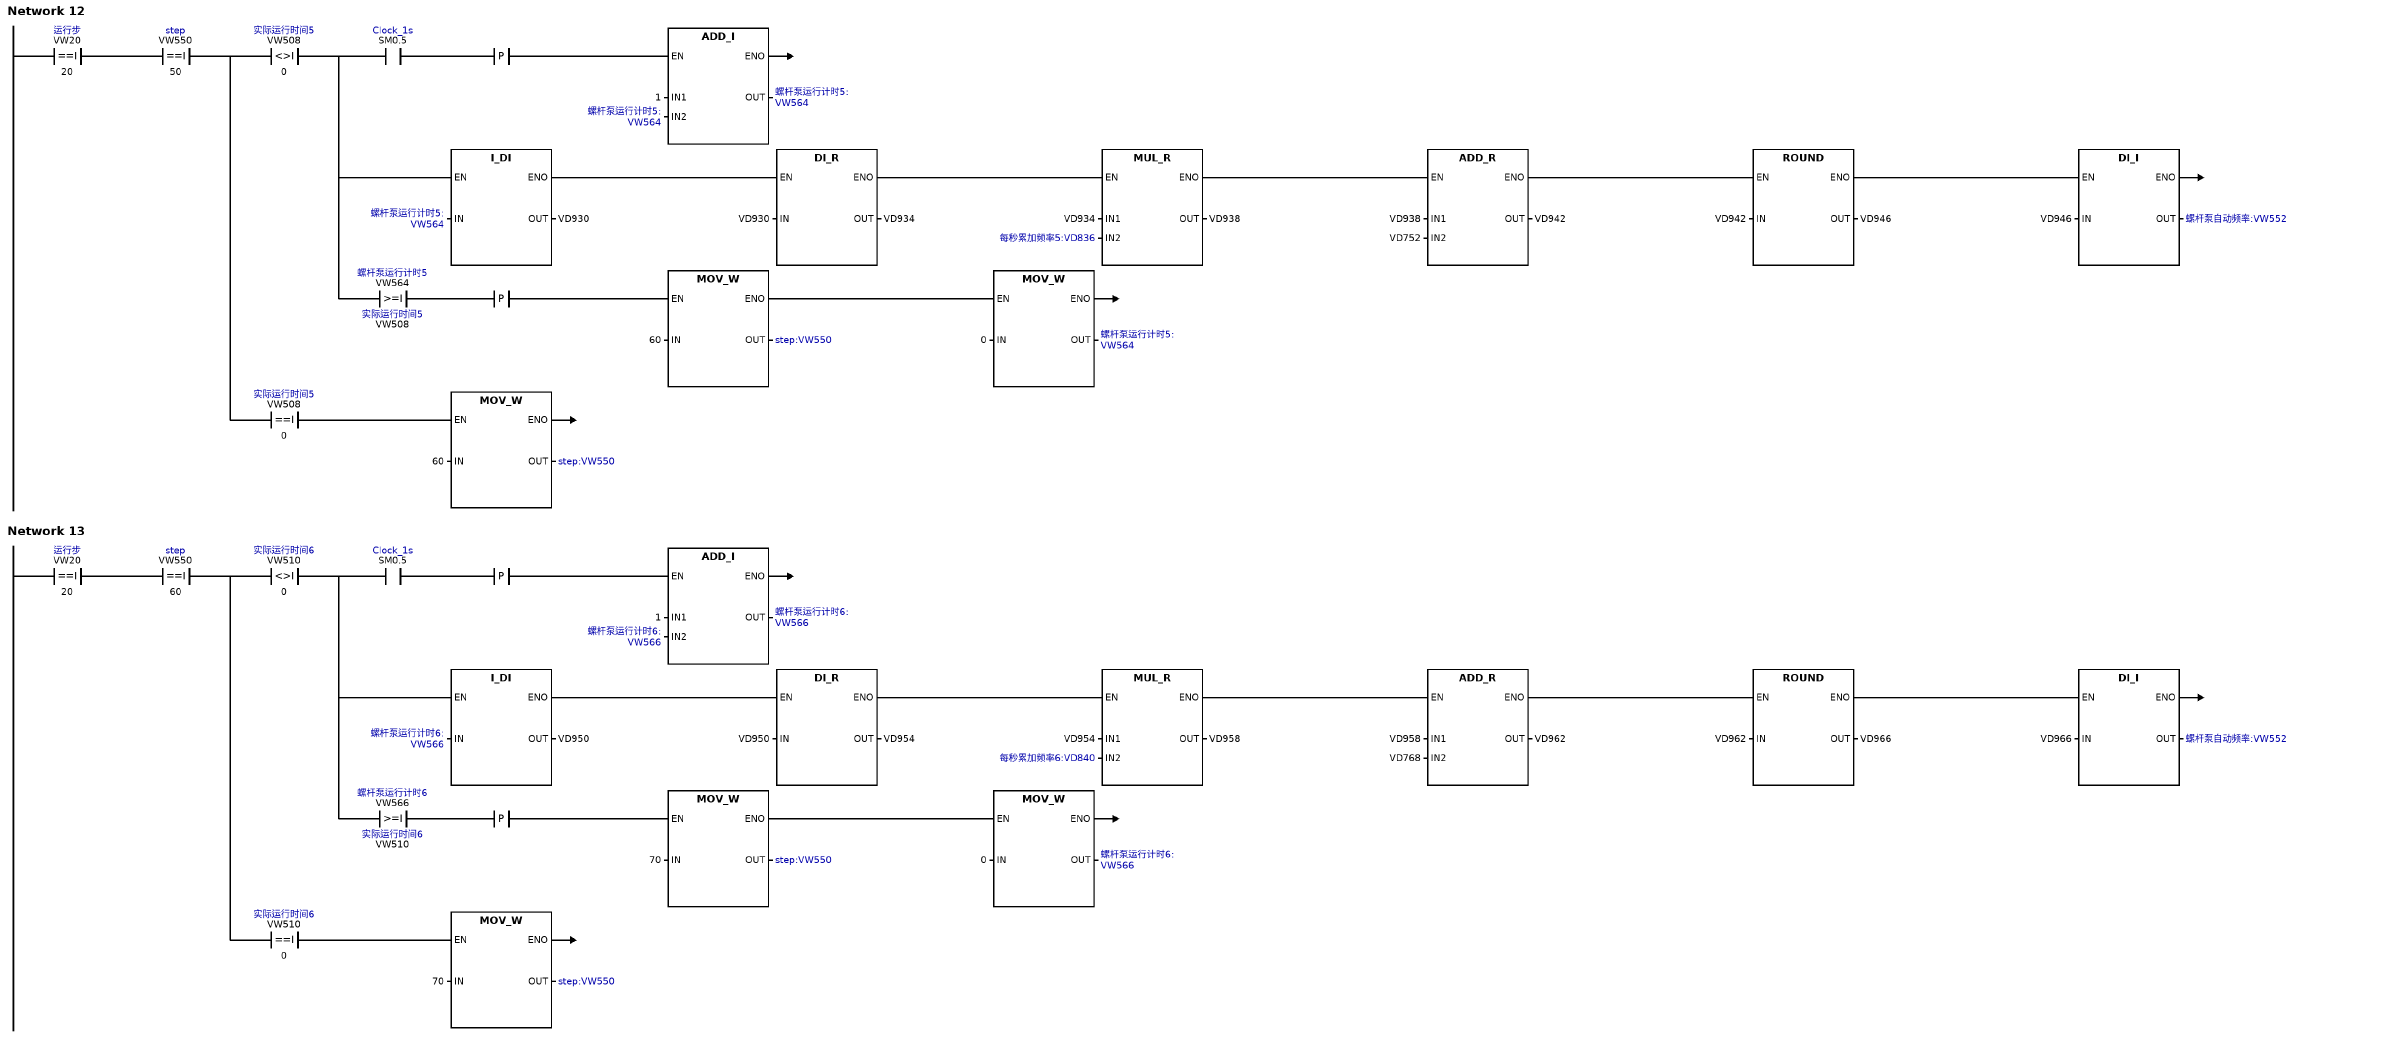
[picture p24: SBR4 networks 12-13]
Network 12
LDW=   运行步:VW20, 20
AW=    step:VW550, 50
LPS
AW<>   实际运行时间5:VW508, 0
LPS
A      Clock_1s:SM0.5
EU
+I     1, 螺杆泵运行计时5:VW564
LRD
ITD    螺杆泵运行计时5:VW564, VD930
AENO
DTR    VD930, VD934
AENO
MOVR   VD934, VD938
AENO
*R     每秒累加频率5:VD836, VD938
AENO
MOVR   VD938, VD942
AENO
+R     VD752, VD942
AENO
ROUND  VD942, VD946
AENO
DTI    VD946, 螺杆泵自动频率:VW552
LPP
AW>=   螺杆泵运行计时5:VW564, 实际运行时间5:VW508
EU
MOVW   60, step:VW550
AENO
MOVW   0, 螺杆泵运行计时5:VW564
LPP
AW=    实际运行时间5:VW508, 0
MOVW   60, step:VW550
Network 13
LDW=   运行步:VW20, 20
AW=    step:VW550, 60
LPS
AW<>   实际运行时间6:VW510, 0
LPS
A      Clock_1s:SM0.5
EU
+I     1, 螺杆泵运行计时6:VW566
LRD
ITD    螺杆泵运行计时6:VW566, VD950
AENO
DTR    VD950, VD954
AENO
MOVR   VD954, VD958
AENO
*R     每秒累加频率6:VD840, VD958
AENO
MOVR   VD958, VD962
AENO
+R     VD768, VD962
AENO
ROUND  VD962, VD966
AENO
DTI    VD966, 螺杆泵自动频率:VW552
LPP
AW>=   螺杆泵运行计时6:VW566, 实际运行时间6:VW510
EU
MOVW   70, step:VW550
AENO
MOVW   0, 螺杆泵运行计时6:VW566
LPP
AW=    实际运行时间6:VW510, 0
MOVW   70, step:VW550
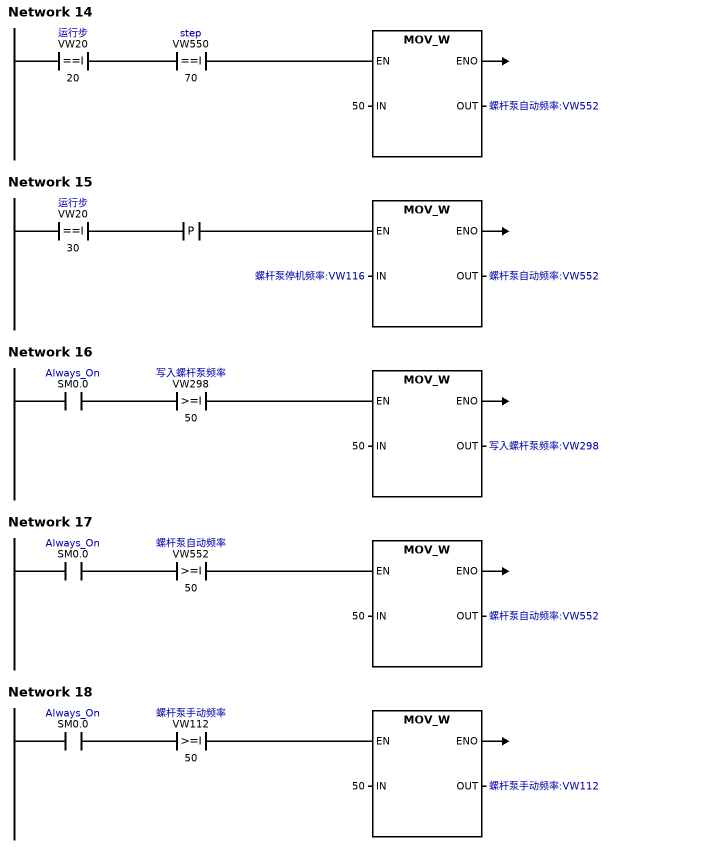
Network 14
LDW=   运行步:VW20, 20
AW=    step:VW550, 70
MOVW   50, 螺杆泵自动频率:VW552
Network 15
LDW=   运行步:VW20, 30
EU
MOVW   螺杆泵停机频率:VW116, 螺杆泵自动频率:VW552
Network 16
LD     Always_On:SM0.0
AW>=   写入螺杆泵频率:VW298, 50
MOVW   50, 写入螺杆泵频率:VW298
Network 17
LD     Always_On:SM0.0
AW>=   螺杆泵自动频率:VW552, 50
MOVW   50, 螺杆泵自动频率:VW552
Network 18
LD     Always_On:SM0.0
AW>=   螺杆泵手动频率:VW112, 50
MOVW   50, 螺杆泵手动频率:VW112
Network 19
// ‘////////////////////////////
END_SUBROUTINE_BLOCK

SUBROUTINE_BLOCK 罗茨泵PID:SBR5
TITLE=子程序注释
BEGIN
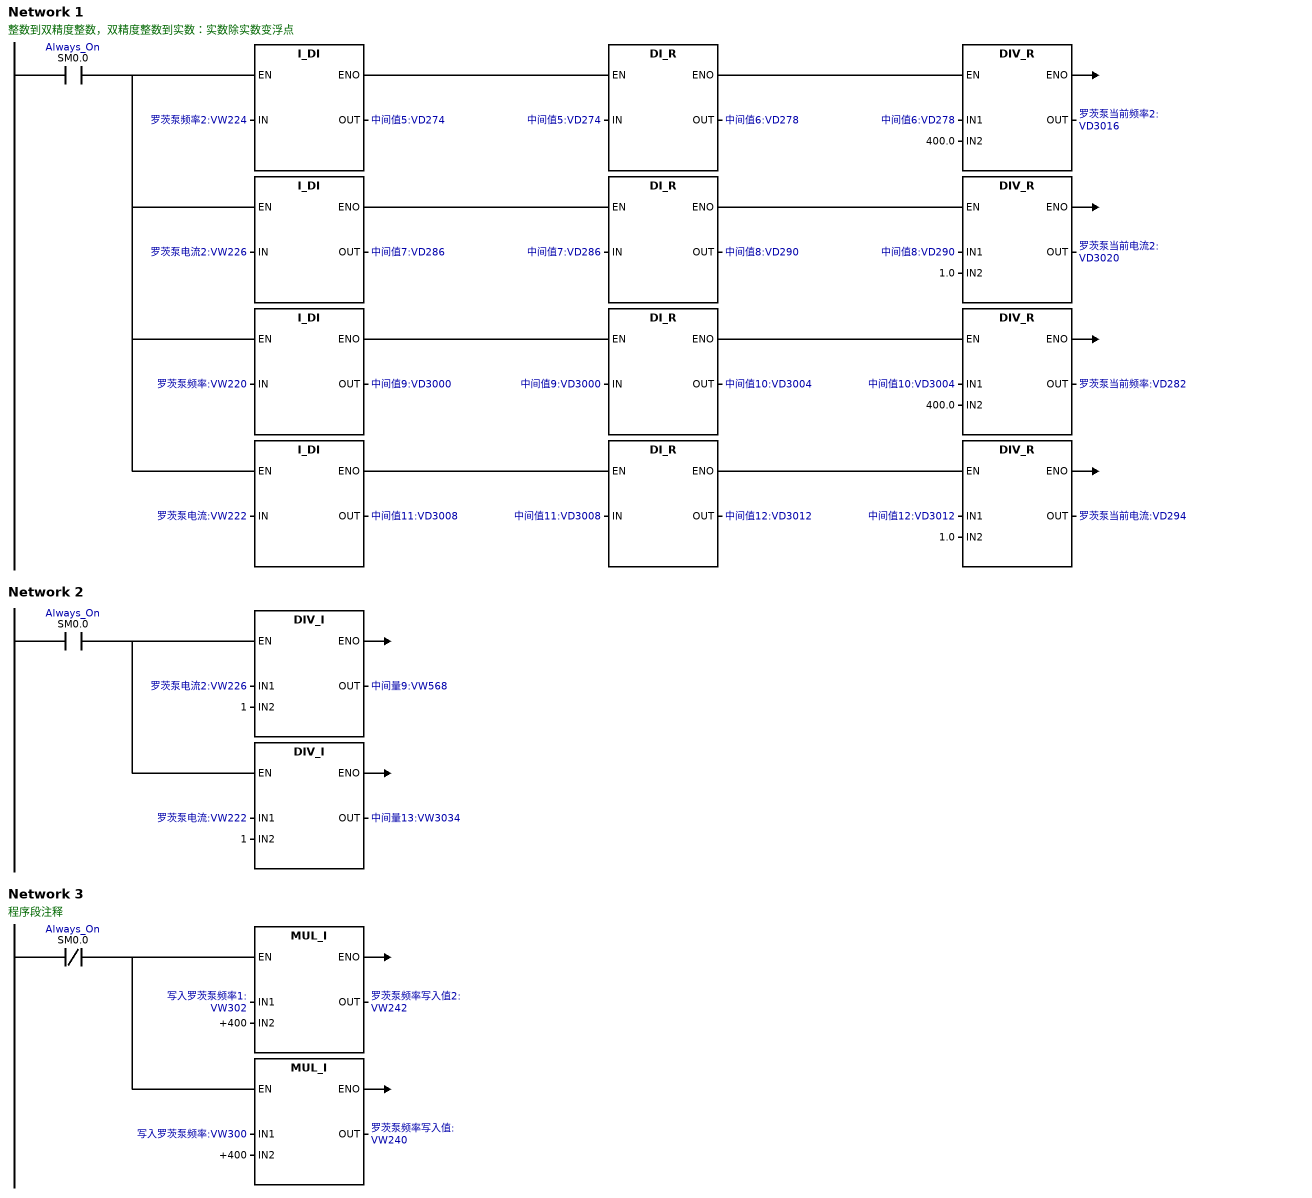
Network 1
// 整数到双精度整数，双精度整数到实数：实数除实数变浮点
LD     Always_On:SM0.0
LPS
ITD    罗茨泵频率2:VW224, 中间值5:VD274
AENO
DTR    中间值5:VD274, 中间值6:VD278
AENO
MOVR   中间值6:VD278, 罗茨泵当前频率2:VD3016
/R     400.0, 罗茨泵当前频率2:VD3016
LRD
ITD    罗茨泵电流2:VW226, 中间值7:VD286
AENO
DTR    中间值7:VD286, 中间值8:VD290
AENO
MOVR   中间值8:VD290, 罗茨泵当前电流2:VD3020
/R     1.0, 罗茨泵当前电流2:VD3020
LRD
ITD    罗茨泵频率:VW220, 中间值9:VD3000
AENO
DTR    中间值9:VD3000, 中间值10:VD3004
AENO
MOVR   中间值10:VD3004, 罗茨泵当前频率:VD282
/R     400.0, 罗茨泵当前频率:VD282
LPP
ITD    罗茨泵电流:VW222, 中间值11:VD3008
AENO
DTR    中间值11:VD3008, 中间值12:VD3012
AENO
MOVR   中间值12:VD3012, 罗茨泵当前电流:VD294
/R     1.0, 罗茨泵当前电流:VD294
Network 2
LD     Always_On:SM0.0
MOVW   罗茨泵电流2:VW226, 中间量9:VW568
/I     1, 中间量9:VW568
MOVW   罗茨泵电流:VW222, 中间量13:VW3034
/I     1, 中间量13:VW3034
Network 3
// 程序段注释
LDN    Always_On:SM0.0
MOVW   写入罗茨泵频率1:VW302, 罗茨泵频率写入值2:VW242
*I     +400, 罗茨泵频率写入值2:VW242
MOVW   写入罗茨泵频率:VW300, 罗茨泵频率写入值:VW240
*I     +400, 罗茨泵频率写入值:VW240
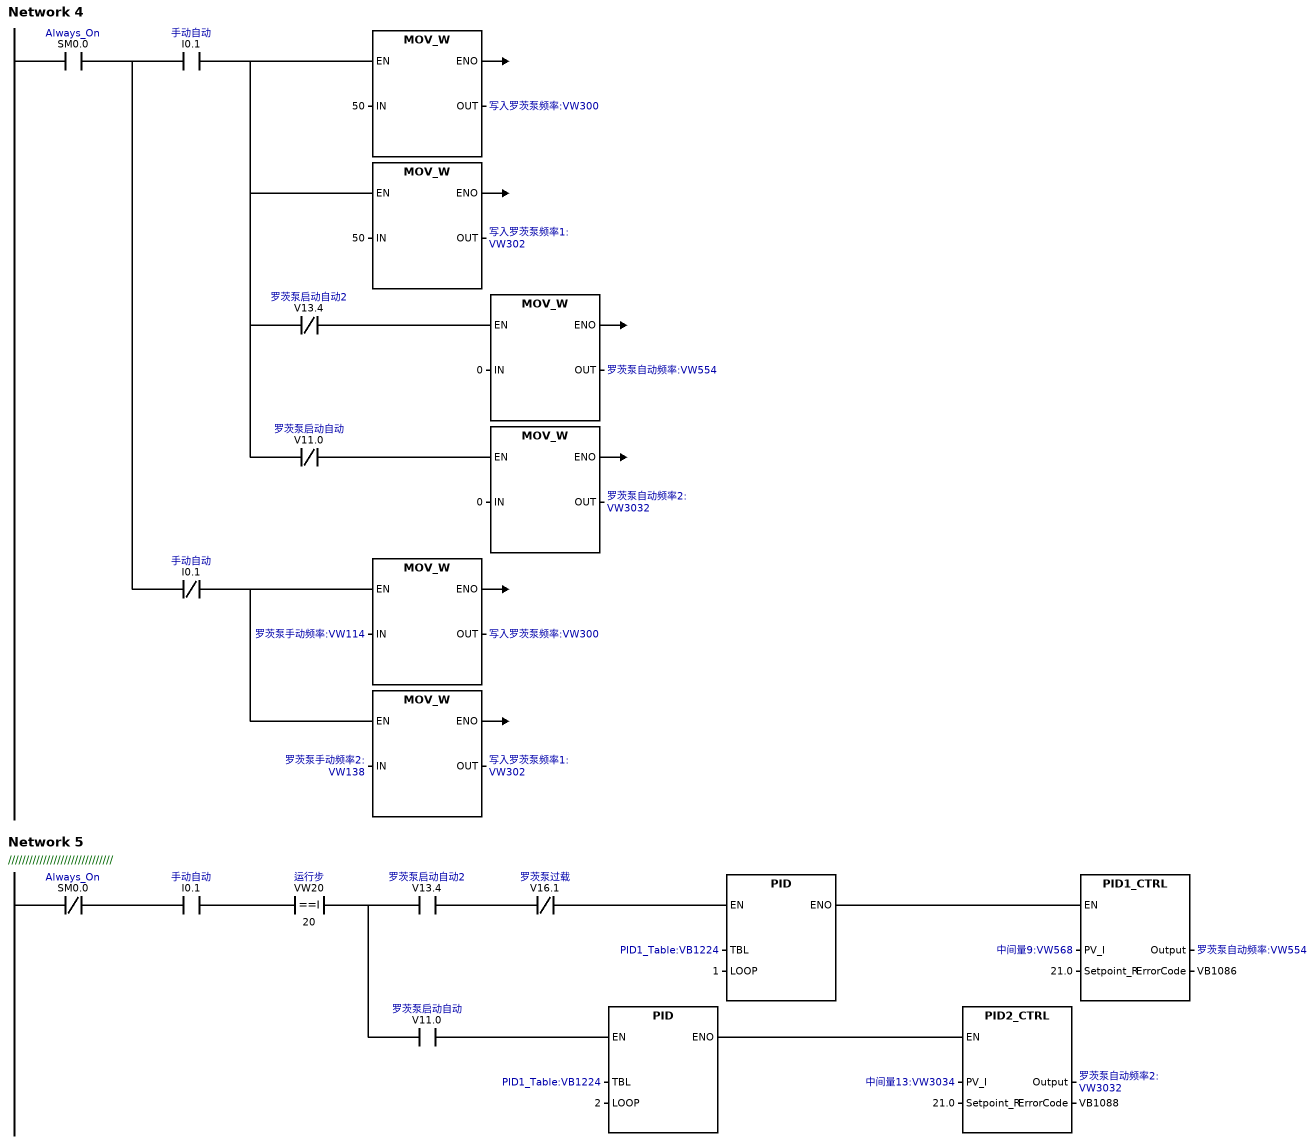
Network 4
LD     Always_On:SM0.0
LPS
A      手动自动:I0.1
LPS
MOVW   50, 写入罗茨泵频率:VW300
MOVW   50, 写入罗茨泵频率1:VW302
AN     罗茨泵启动自动2:V13.4
MOVW   0, 罗茨泵自动频率:VW554
LPP
AN     罗茨泵启动自动:V11.0
MOVW   0, 罗茨泵自动频率2:VW3032
LPP
AN     手动自动:I0.1
MOVW   罗茨泵手动频率:VW114, 写入罗茨泵频率:VW300
MOVW   罗茨泵手动频率2:VW138, 写入罗茨泵频率1:VW302
Network 5
// //////////////////////////////
LDN    Always_On:SM0.0
A      手动自动:I0.1
AW=    运行步:VW20, 20
LPS
A      罗茨泵启动自动2:V13.4
AN     罗茨泵过载:V16.1
PID    PID1_Table:VB1224, 1
AENO
CALL   PID1_CTRL:SBR16, 中间量9:VW568, 21.0, 罗茨泵自动频率:VW554, VB1086
LPP
A      罗茨泵启动自动:V11.0
PID    PID1_Table:VB1224, 2
AENO
CALL   PID2_CTRL:SBR17, 中间量13:VW3034, 21.0, 罗茨泵自动频率2:VW3032, VB1088
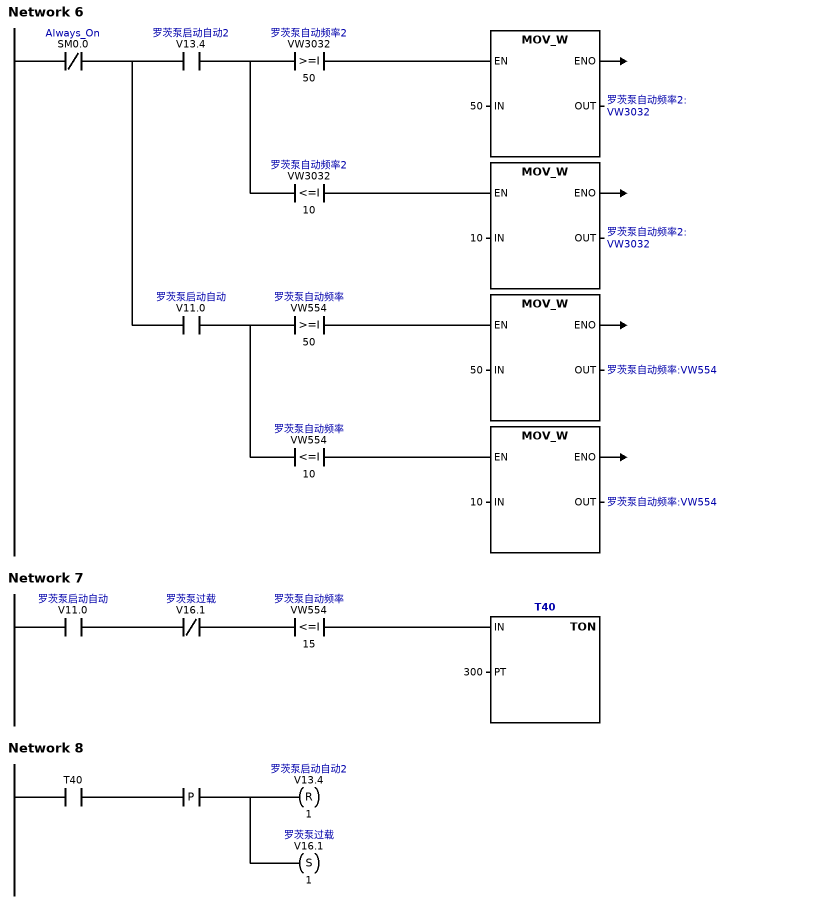
Network 6
LDN    Always_On:SM0.0
LPS
A      罗茨泵启动自动2:V13.4
LPS
AW>=   罗茨泵自动频率2:VW3032, 50
MOVW   50, 罗茨泵自动频率2:VW3032
LPP
AW<=   罗茨泵自动频率2:VW3032, 10
MOVW   10, 罗茨泵自动频率2:VW3032
LPP
A      罗茨泵启动自动:V11.0
LPS
AW>=   罗茨泵自动频率:VW554, 50
MOVW   50, 罗茨泵自动频率:VW554
LPP
AW<=   罗茨泵自动频率:VW554, 10
MOVW   10, 罗茨泵自动频率:VW554
Network 7
LD     罗茨泵启动自动:V11.0
AN     罗茨泵过载:V16.1
AW<=   罗茨泵自动频率:VW554, 15
TON    T40, 300
Network 8
LD     T40
EU
R      罗茨泵启动自动2:V13.4, 1
S      罗茨泵过载:V16.1, 1
END_SUBROUTINE_BLOCK

SUBROUTINE_BLOCK 报警:SBR6
TITLE=子程序注释
BEGIN
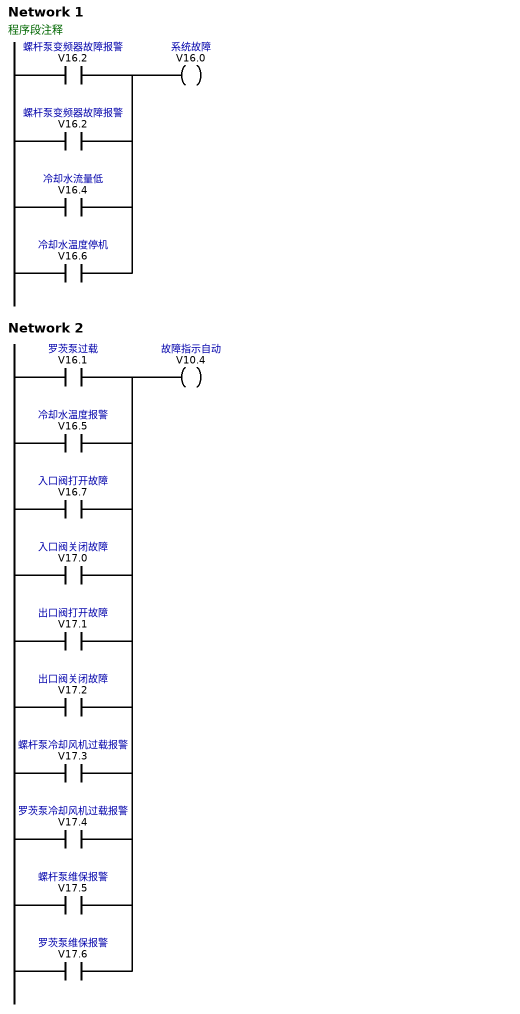
Network 1
// 程序段注释
LD     螺杆泵变频器故障报警:V16.2
O      螺杆泵变频器故障报警:V16.2
O      冷却水流量低:V16.4
O      冷却水温度停机:V16.6
=      系统故障:V16.0
Network 2
LD     罗茨泵过载:V16.1
O      冷却水温度报警:V16.5
O      入口阀打开故障:V16.7
O      入口阀关闭故障:V17.0
O      出口阀打开故障:V17.1
O      出口阀关闭故障:V17.2
O      螺杆泵冷却风机过载报警:V17.3
O      罗茨泵冷却风机过载报警:V17.4
O      螺杆泵维保报警:V17.5
O      罗茨泵维保报警:V17.6
=      故障指示自动:V10.4
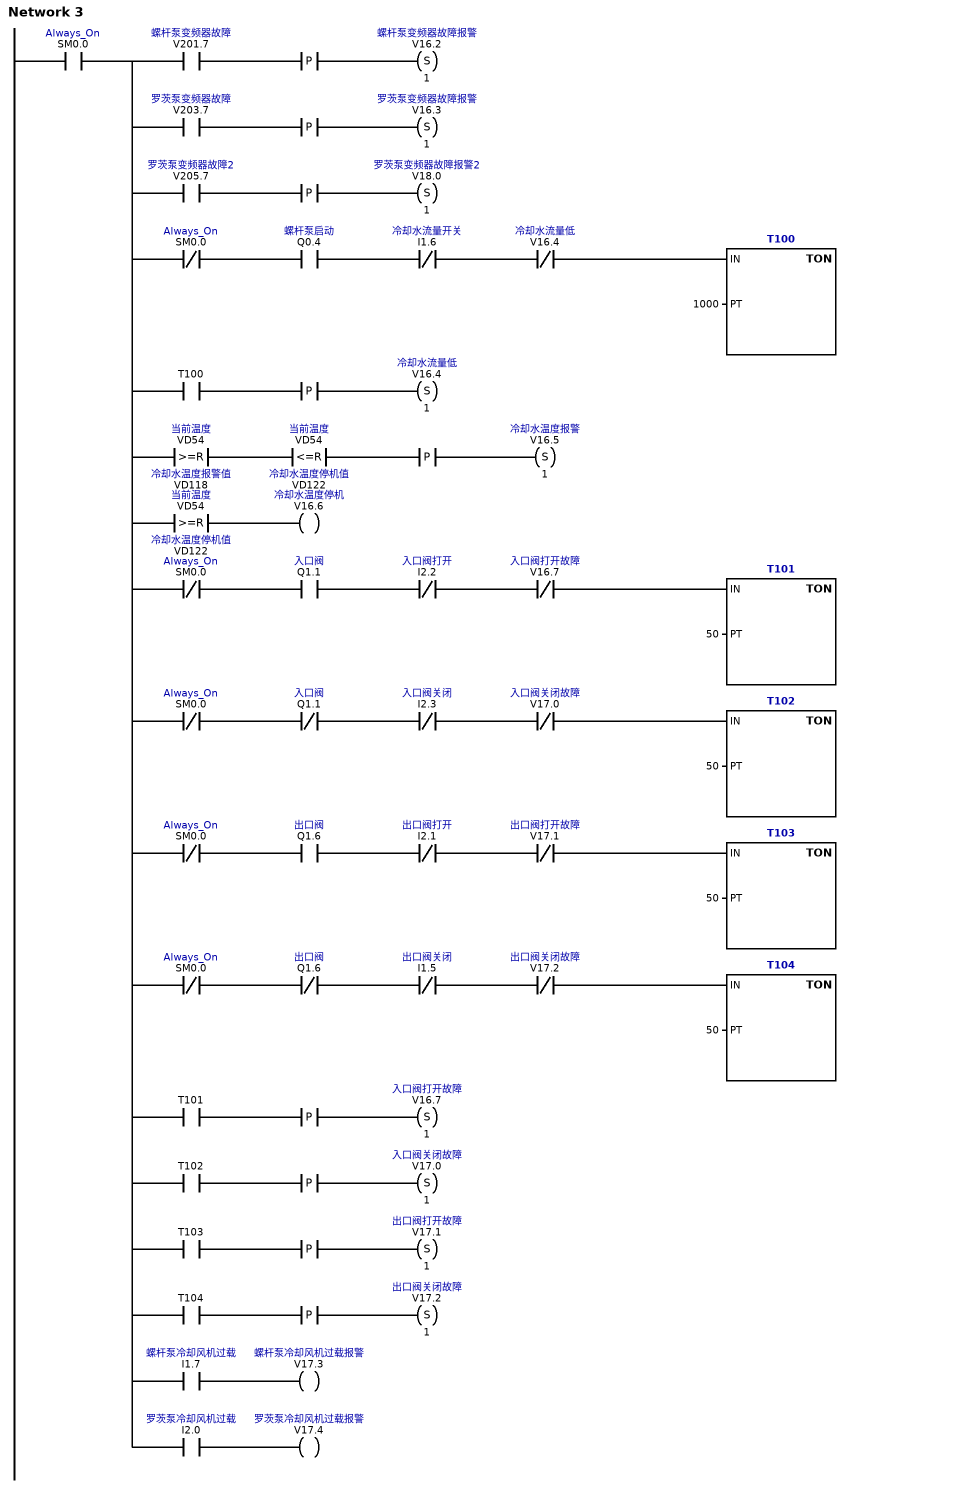
Network 3
LD     Always_On:SM0.0
LPS
A      螺杆泵变频器故障:V201.7
EU
S      螺杆泵变频器故障报警:V16.2, 1
LRD
A      罗茨泵变频器故障:V203.7
EU
S      罗茨泵变频器故障报警:V16.3, 1
LRD
A      罗茨泵变频器故障2:V205.7
EU
S      罗茨泵变频器故障报警2:V18.0, 1
LRD
AN     Always_On:SM0.0
A      螺杆泵启动:Q0.4
AN     冷却水流量开关:I1.6
AN     冷却水流量低:V16.4
TON    T100, 1000
LRD
A      T100
EU
S      冷却水流量低:V16.4, 1
LRD
AR>=   当前温度:VD54, 冷却水温度报警值:VD118
AR<=   当前温度:VD54, 冷却水温度停机值:VD122
EU
S      冷却水温度报警:V16.5, 1
LRD
AR>=   当前温度:VD54, 冷却水温度停机值:VD122
=      冷却水温度停机:V16.6
LRD
AN     Always_On:SM0.0
A      入口阀:Q1.1
AN     入口阀打开:I2.2
AN     入口阀打开故障:V16.7
TON    T101, 50
LRD
AN     Always_On:SM0.0
AN     入口阀:Q1.1
AN     入口阀关闭:I2.3
AN     入口阀关闭故障:V17.0
TON    T102, 50
LRD
AN     Always_On:SM0.0
A      出口阀:Q1.6
AN     出口阀打开:I2.1
AN     出口阀打开故障:V17.1
TON    T103, 50
LRD
AN     Always_On:SM0.0
AN     出口阀:Q1.6
AN     出口阀关闭:I1.5
AN     出口阀关闭故障:V17.2
TON    T104, 50
LRD
A      T101
EU
S      入口阀打开故障:V16.7, 1
LRD
A      T102
EU
S      入口阀关闭故障:V17.0, 1
LRD
A      T103
EU
S      出口阀打开故障:V17.1, 1
LRD
A      T104
EU
S      出口阀关闭故障:V17.2, 1
LRD
A      螺杆泵冷却风机过载:I1.7
=      螺杆泵冷却风机过载报警:V17.3
LPP
A      罗茨泵冷却风机过载:I2.0
=      罗茨泵冷却风机过载报警:V17.4
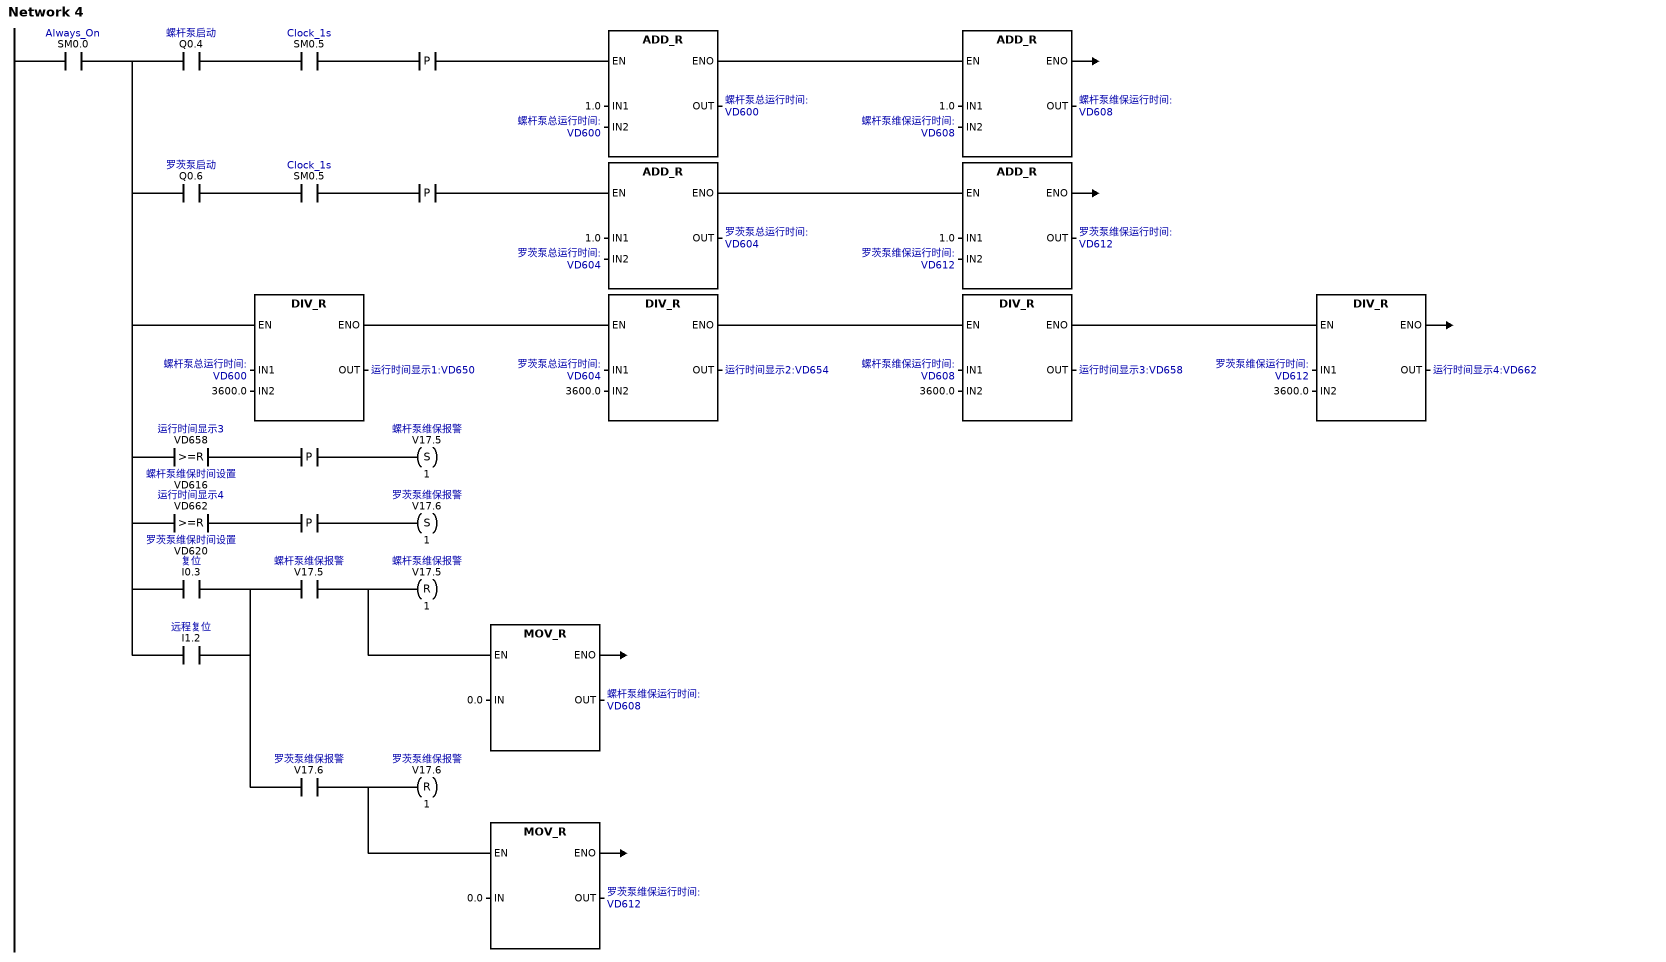
Network 4
LD     Always_On:SM0.0
LPS
A      螺杆泵启动:Q0.4
A      Clock_1s:SM0.5
EU
+R     1.0, 螺杆泵总运行时间:VD600
AENO
+R     1.0, 螺杆泵维保运行时间:VD608
LRD
A      罗茨泵启动:Q0.6
A      Clock_1s:SM0.5
EU
+R     1.0, 罗茨泵总运行时间:VD604
AENO
+R     1.0, 罗茨泵维保运行时间:VD612
LRD
MOVR   螺杆泵总运行时间:VD600, 运行时间显示1:VD650
AENO
/R     3600.0, 运行时间显示1:VD650
AENO
MOVR   罗茨泵总运行时间:VD604, 运行时间显示2:VD654
AENO
/R     3600.0, 运行时间显示2:VD654
AENO
MOVR   螺杆泵维保运行时间:VD608, 运行时间显示3:VD658
AENO
/R     3600.0, 运行时间显示3:VD658
AENO
MOVR   罗茨泵维保运行时间:VD612, 运行时间显示4:VD662
/R     3600.0, 运行时间显示4:VD662
LRD
AR>=   运行时间显示3:VD658, 螺杆泵维保时间设置:VD616
EU
S      螺杆泵维保报警:V17.5, 1
LRD
AR>=   运行时间显示4:VD662, 罗茨泵维保时间设置:VD620
EU
S      罗茨泵维保报警:V17.6, 1
LPP
LD     复位:I0.3
O      远程复位:I1.2
ALD
LPS
A      螺杆泵维保报警:V17.5
R      螺杆泵维保报警:V17.5, 1
MOVR   0.0, 螺杆泵维保运行时间:VD608
LPP
A      罗茨泵维保报警:V17.6
R      罗茨泵维保报警:V17.6, 1
MOVR   0.0, 罗茨泵维保运行时间:VD612
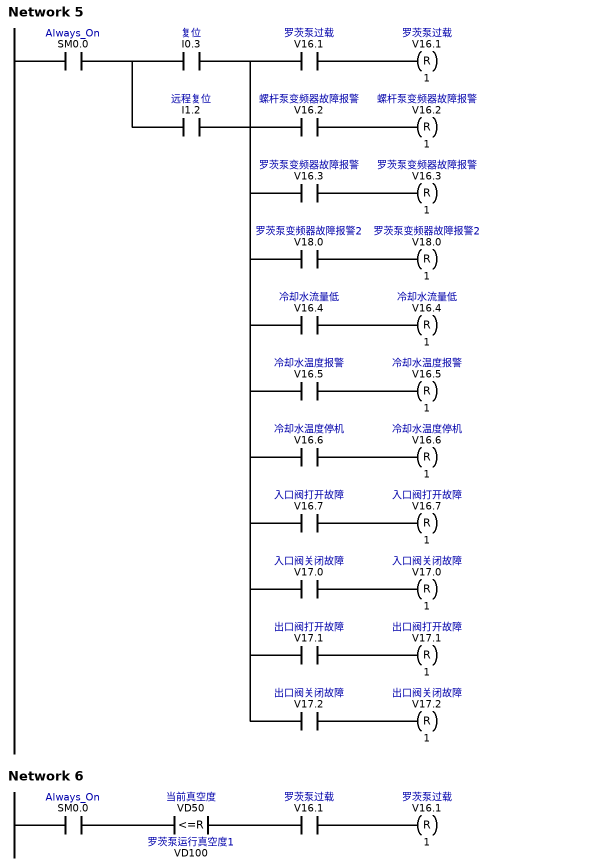
Network 5
LD     Always_On:SM0.0
LD     复位:I0.3
O      远程复位:I1.2
ALD
LPS
A      罗茨泵过载:V16.1
R      罗茨泵过载:V16.1, 1
LRD
A      螺杆泵变频器故障报警:V16.2
R      螺杆泵变频器故障报警:V16.2, 1
LRD
A      罗茨泵变频器故障报警:V16.3
R      罗茨泵变频器故障报警:V16.3, 1
LRD
A      罗茨泵变频器故障报警2:V18.0
R      罗茨泵变频器故障报警2:V18.0, 1
LRD
A      冷却水流量低:V16.4
R      冷却水流量低:V16.4, 1
LRD
A      冷却水温度报警:V16.5
R      冷却水温度报警:V16.5, 1
LRD
A      冷却水温度停机:V16.6
R      冷却水温度停机:V16.6, 1
LRD
A      入口阀打开故障:V16.7
R      入口阀打开故障:V16.7, 1
LRD
A      入口阀关闭故障:V17.0
R      入口阀关闭故障:V17.0, 1
LRD
A      出口阀打开故障:V17.1
R      出口阀打开故障:V17.1, 1
LPP
A      出口阀关闭故障:V17.2
R      出口阀关闭故障:V17.2, 1
Network 6
LD     Always_On:SM0.0
AR<=   当前真空度:VD50, 罗茨泵运行真空度1:VD100
A      罗茨泵过载:V16.1
R      罗茨泵过载:V16.1, 1
END_SUBROUTINE_BLOCK

// SBR7: protected block, not included

// SBR8: protected block, not included

// SBR9: protected block, not included

// SBR10: protected block, not included

SUBROUTINE_BLOCK DCS:SBR11
TITLE=子程序注释
BEGIN
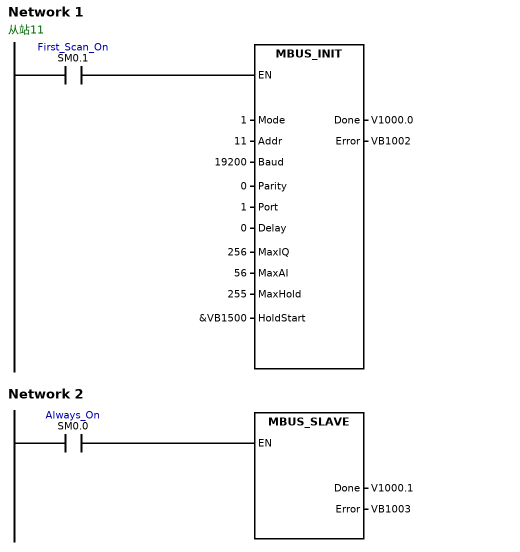
Network 1
// 从站11
LD     First_Scan_On:SM0.1
CALL   MBUS_INIT:SBR12, 1, 11, 19200, 0, 1, 0, 256, 56, 255, &VB1500, V1000.0, VB1002
Network 2
LD     Always_On:SM0.0
CALL   MBUS_SLAVE:SBR13, V1000.1, VB1003
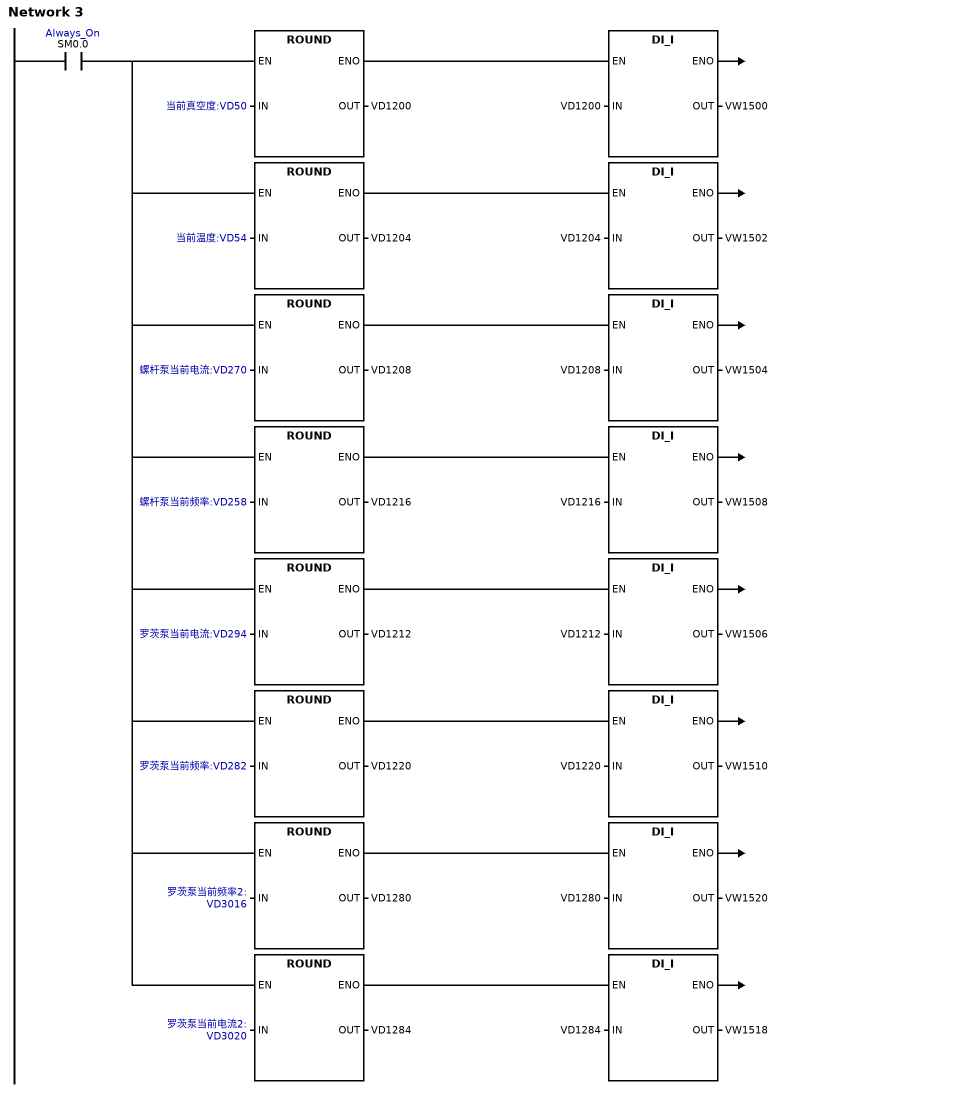
Network 3
LD     Always_On:SM0.0
LPS
ROUND  当前真空度:VD50, VD1200
AENO
DTI    VD1200, VW1500
LRD
ROUND  当前温度:VD54, VD1204
AENO
DTI    VD1204, VW1502
LRD
ROUND  螺杆泵当前电流:VD270, VD1208
AENO
DTI    VD1208, VW1504
LRD
ROUND  螺杆泵当前频率:VD258, VD1216
AENO
DTI    VD1216, VW1508
LRD
ROUND  罗茨泵当前电流:VD294, VD1212
AENO
DTI    VD1212, VW1506
LRD
ROUND  罗茨泵当前频率:VD282, VD1220
AENO
DTI    VD1220, VW1510
LRD
ROUND  罗茨泵当前频率2:VD3016, VD1280
AENO
DTI    VD1280, VW1520
LPP
ROUND  罗茨泵当前电流2:VD3020, VD1284
AENO
DTI    VD1284, VW1518
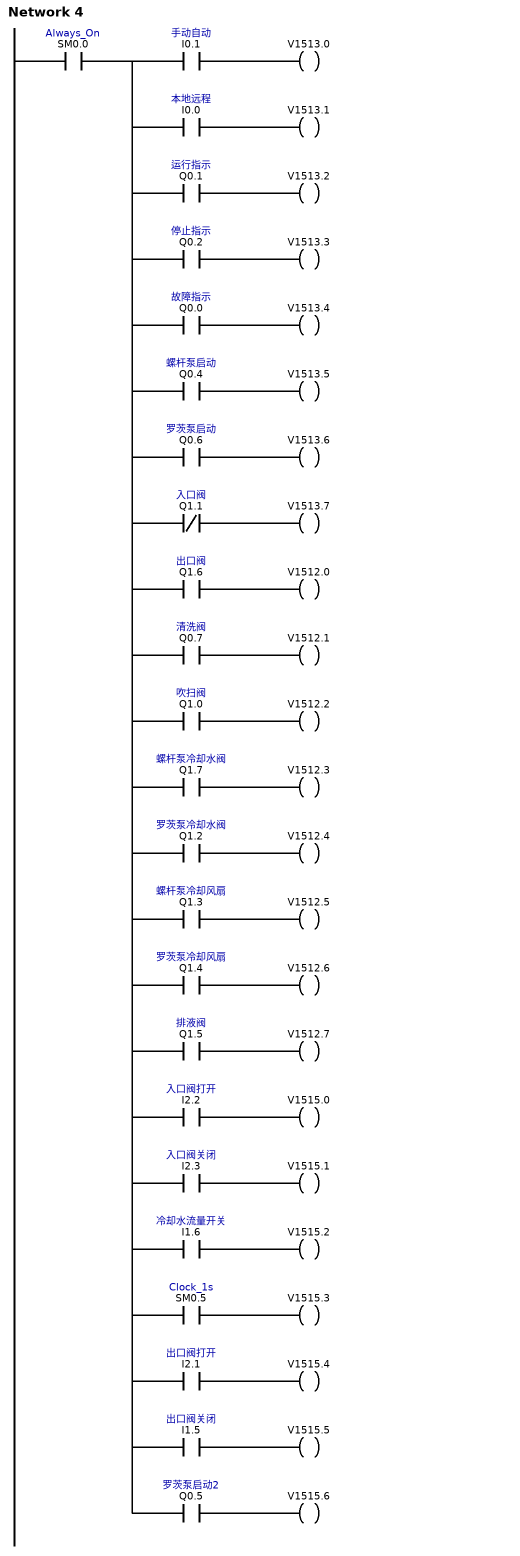
Network 4
LD     Always_On:SM0.0
LPS
A      手动自动:I0.1
=      V1513.0
LRD
A      本地远程:I0.0
=      V1513.1
LRD
A      运行指示:Q0.1
=      V1513.2
LRD
A      停止指示:Q0.2
=      V1513.3
LRD
A      故障指示:Q0.0
=      V1513.4
LRD
A      螺杆泵启动:Q0.4
=      V1513.5
LRD
A      罗茨泵启动:Q0.6
=      V1513.6
LRD
AN     入口阀:Q1.1
=      V1513.7
LRD
A      出口阀:Q1.6
=      V1512.0
LRD
A      清洗阀:Q0.7
=      V1512.1
LRD
A      吹扫阀:Q1.0
=      V1512.2
LRD
A      螺杆泵冷却水阀:Q1.7
=      V1512.3
LRD
A      罗茨泵冷却水阀:Q1.2
=      V1512.4
LRD
A      螺杆泵冷却风扇:Q1.3
=      V1512.5
LRD
A      罗茨泵冷却风扇:Q1.4
=      V1512.6
LRD
A      排液阀:Q1.5
=      V1512.7
LRD
A      入口阀打开:I2.2
=      V1515.0
LRD
A      入口阀关闭:I2.3
=      V1515.1
LRD
A      冷却水流量开关:I1.6
=      V1515.2
LRD
A      Clock_1s:SM0.5
=      V1515.3
LRD
A      出口阀打开:I2.1
=      V1515.4
LRD
A      出口阀关闭:I1.5
=      V1515.5
LPP
A      罗茨泵启动2:Q0.5
=      V1515.6
END_SUBROUTINE_BLOCK

// SBR12: protected block, not included

// SBR13: protected block, not included

// SBR14: protected block, not included

SUBROUTINE_BLOCK 螺杆泵新配方稳压:SBR15
TITLE=子程序注释
BEGIN
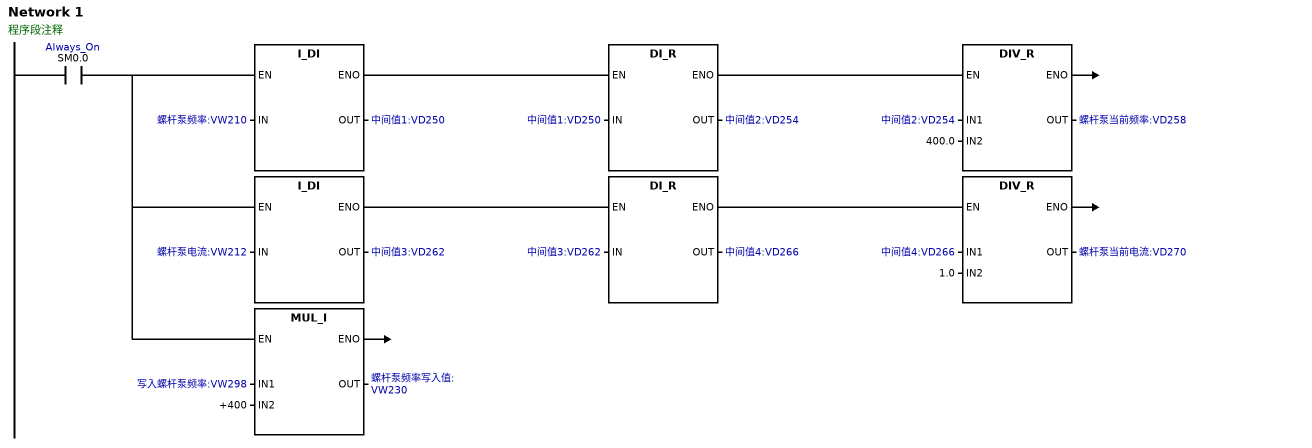
Network 1
// 程序段注释
LD     Always_On:SM0.0
LPS
ITD    螺杆泵频率:VW210, 中间值1:VD250
AENO
DTR    中间值1:VD250, 中间值2:VD254
AENO
MOVR   中间值2:VD254, 螺杆泵当前频率:VD258
/R     400.0, 螺杆泵当前频率:VD258
LRD
ITD    螺杆泵电流:VW212, 中间值3:VD262
AENO
DTR    中间值3:VD262, 中间值4:VD266
AENO
MOVR   中间值4:VD266, 螺杆泵当前电流:VD270
/R     1.0, 螺杆泵当前电流:VD270
LPP
MOVW   写入螺杆泵频率:VW298, 螺杆泵频率写入值:VW230
*I     +400, 螺杆泵频率写入值:VW230
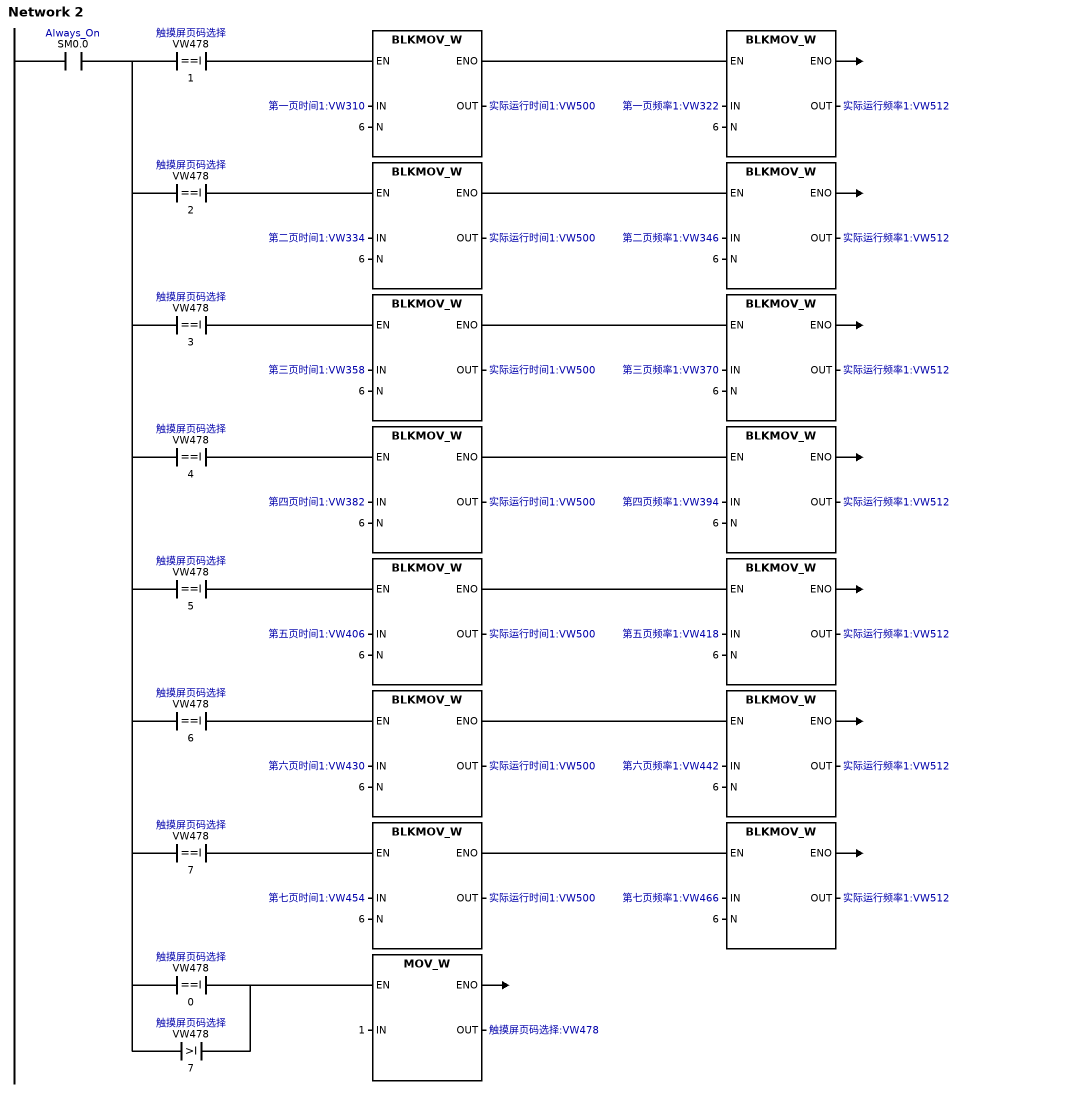
Network 2
LD     Always_On:SM0.0
LPS
AW=    触摸屏页码选择:VW478, 1
BMW    第一页时间1:VW310, 实际运行时间1:VW500, 6
AENO
BMW    第一页频率1:VW322, 实际运行频率1:VW512, 6
LRD
AW=    触摸屏页码选择:VW478, 2
BMW    第二页时间1:VW334, 实际运行时间1:VW500, 6
AENO
BMW    第二页频率1:VW346, 实际运行频率1:VW512, 6
LRD
AW=    触摸屏页码选择:VW478, 3
BMW    第三页时间1:VW358, 实际运行时间1:VW500, 6
AENO
BMW    第三页频率1:VW370, 实际运行频率1:VW512, 6
LRD
AW=    触摸屏页码选择:VW478, 4
BMW    第四页时间1:VW382, 实际运行时间1:VW500, 6
AENO
BMW    第四页频率1:VW394, 实际运行频率1:VW512, 6
LRD
AW=    触摸屏页码选择:VW478, 5
BMW    第五页时间1:VW406, 实际运行时间1:VW500, 6
AENO
BMW    第五页频率1:VW418, 实际运行频率1:VW512, 6
LRD
AW=    触摸屏页码选择:VW478, 6
BMW    第六页时间1:VW430, 实际运行时间1:VW500, 6
AENO
BMW    第六页频率1:VW442, 实际运行频率1:VW512, 6
LRD
AW=    触摸屏页码选择:VW478, 7
BMW    第七页时间1:VW454, 实际运行时间1:VW500, 6
AENO
BMW    第七页频率1:VW466, 实际运行频率1:VW512, 6
LPP
LDW=   触摸屏页码选择:VW478, 0
OW>    触摸屏页码选择:VW478, 7
ALD
MOVW   1, 触摸屏页码选择:VW478
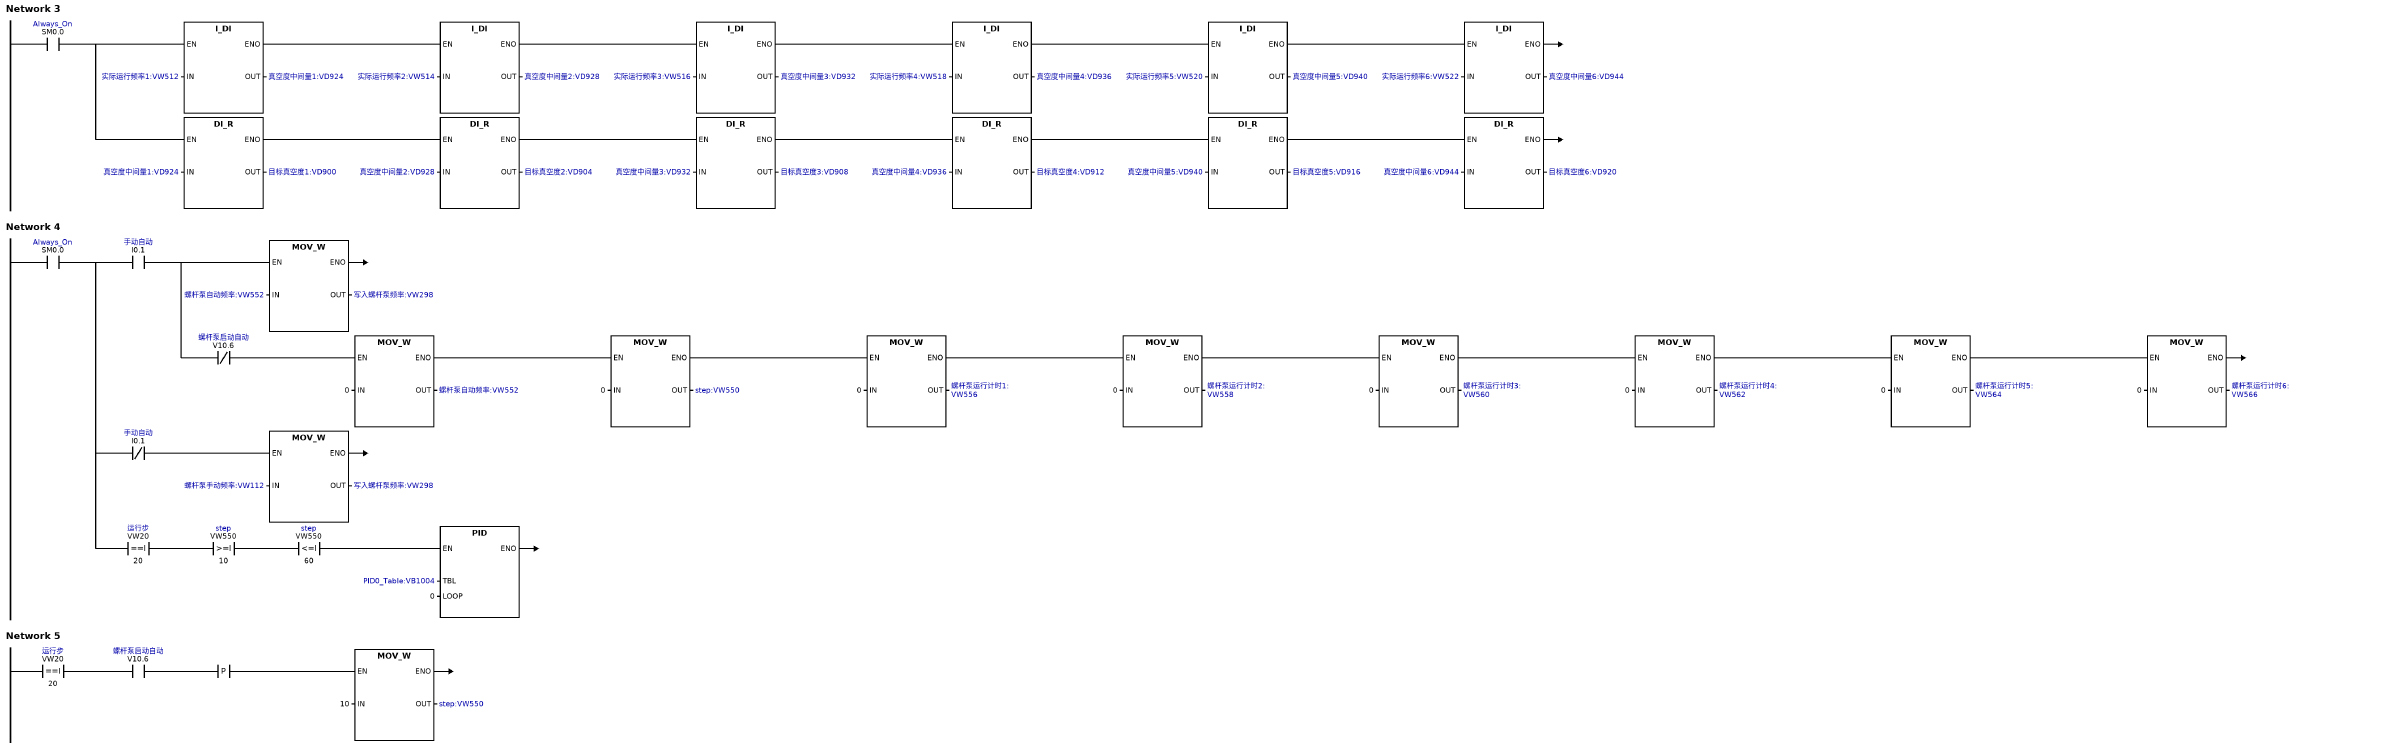
Network 3
LD     Always_On:SM0.0
LPS
ITD    实际运行频率1:VW512, 真空度中间量1:VD924
AENO
ITD    实际运行频率2:VW514, 真空度中间量2:VD928
AENO
ITD    实际运行频率3:VW516, 真空度中间量3:VD932
AENO
ITD    实际运行频率4:VW518, 真空度中间量4:VD936
AENO
ITD    实际运行频率5:VW520, 真空度中间量5:VD940
AENO
ITD    实际运行频率6:VW522, 真空度中间量6:VD944
LPP
DTR    真空度中间量1:VD924, 目标真空度1:VD900
AENO
DTR    真空度中间量2:VD928, 目标真空度2:VD904
AENO
DTR    真空度中间量3:VD932, 目标真空度3:VD908
AENO
DTR    真空度中间量4:VD936, 目标真空度4:VD912
AENO
DTR    真空度中间量5:VD940, 目标真空度5:VD916
AENO
DTR    真空度中间量6:VD944, 目标真空度6:VD920
Network 4
LD     Always_On:SM0.0
LPS
A      手动自动:I0.1
MOVW   螺杆泵自动频率:VW552, 写入螺杆泵频率:VW298
AN     螺杆泵启动自动:V10.6
MOVW   0, 螺杆泵自动频率:VW552
AENO
MOVW   0, step:VW550
AENO
MOVW   0, 螺杆泵运行计时1:VW556
AENO
MOVW   0, 螺杆泵运行计时2:VW558
AENO
MOVW   0, 螺杆泵运行计时3:VW560
AENO
MOVW   0, 螺杆泵运行计时4:VW562
AENO
MOVW   0, 螺杆泵运行计时5:VW564
AENO
MOVW   0, 螺杆泵运行计时6:VW566
LPP
LPS
AN     手动自动:I0.1
MOVW   螺杆泵手动频率:VW112, 写入螺杆泵频率:VW298
LPP
AW=    运行步:VW20, 20
AW>=   step:VW550, 10
AW<=   step:VW550, 60
PID    PID0_Table:VB1004, 0
Network 5
LDW=   运行步:VW20, 20
A      螺杆泵启动自动:V10.6
EU
MOVW   10, step:VW550
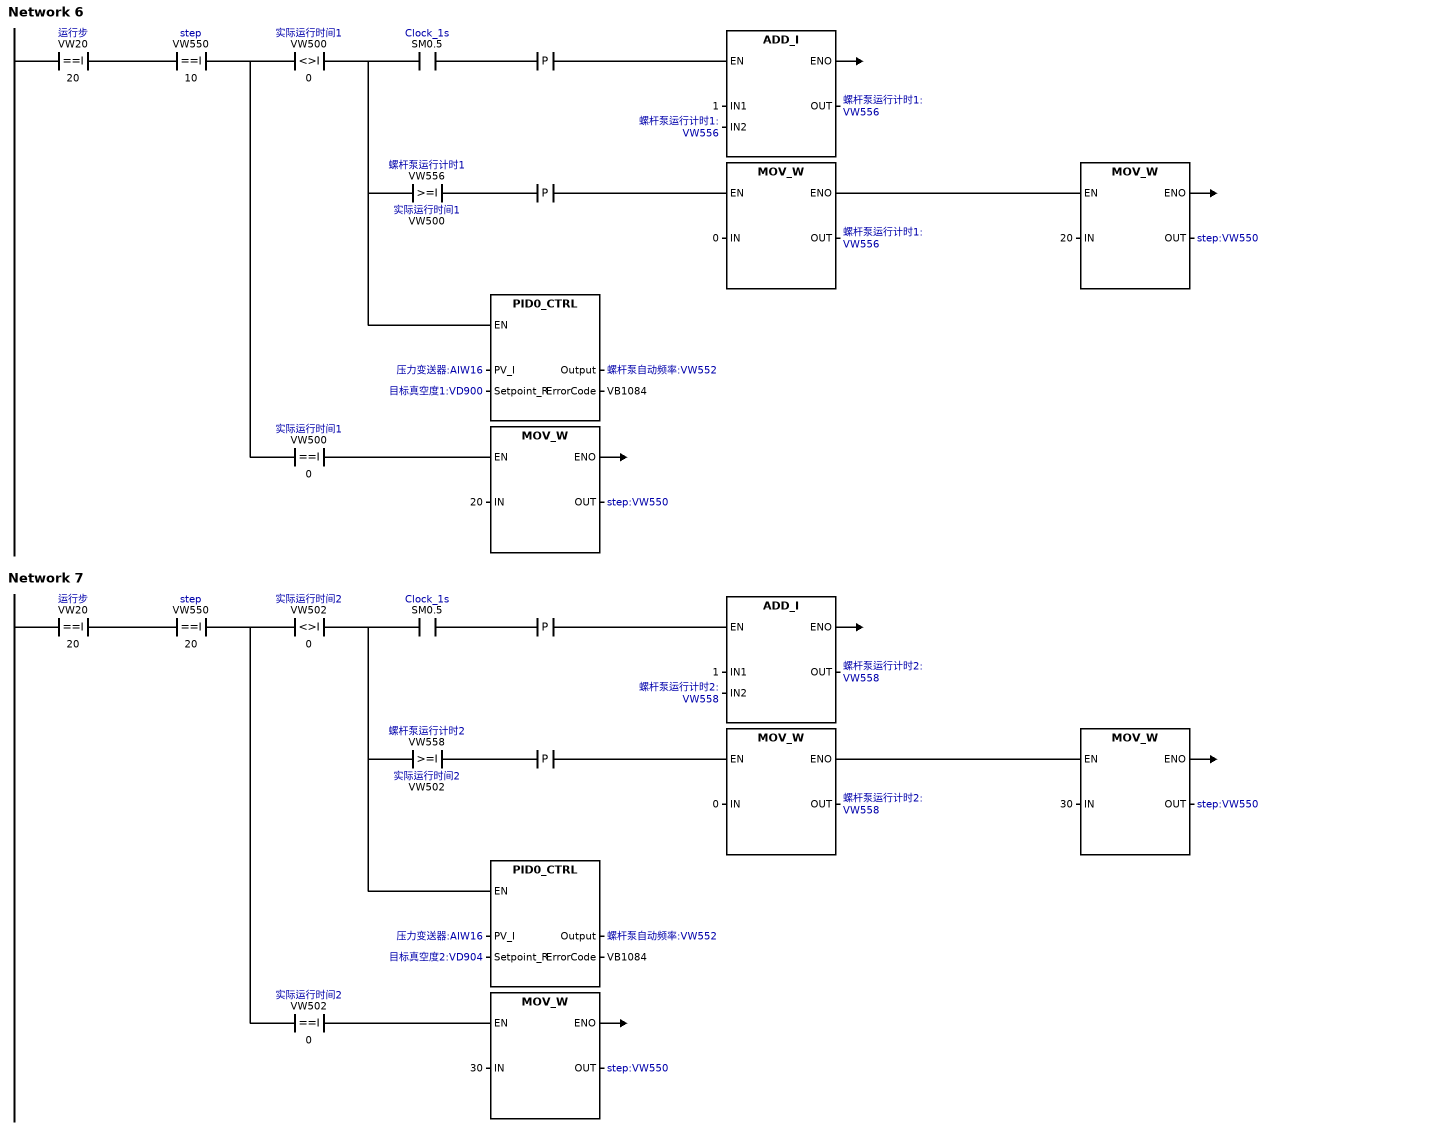
Network 6
LDW=   运行步:VW20, 20
AW=    step:VW550, 10
LPS
AW<>   实际运行时间1:VW500, 0
LPS
A      Clock_1s:SM0.5
EU
+I     1, 螺杆泵运行计时1:VW556
LRD
AW>=   螺杆泵运行计时1:VW556, 实际运行时间1:VW500
EU
MOVW   0, 螺杆泵运行计时1:VW556
AENO
MOVW   20, step:VW550
LPP
CALL   PID0_CTRL:SBR10, 压力变送器:AIW16, 目标真空度1:VD900, 螺杆泵自动频率:VW552, VB1084
LPP
AW=    实际运行时间1:VW500, 0
MOVW   20, step:VW550
Network 7
LDW=   运行步:VW20, 20
AW=    step:VW550, 20
LPS
AW<>   实际运行时间2:VW502, 0
LPS
A      Clock_1s:SM0.5
EU
+I     1, 螺杆泵运行计时2:VW558
LRD
AW>=   螺杆泵运行计时2:VW558, 实际运行时间2:VW502
EU
MOVW   0, 螺杆泵运行计时2:VW558
AENO
MOVW   30, step:VW550
LPP
CALL   PID0_CTRL:SBR10, 压力变送器:AIW16, 目标真空度2:VD904, 螺杆泵自动频率:VW552, VB1084
LPP
AW=    实际运行时间2:VW502, 0
MOVW   30, step:VW550
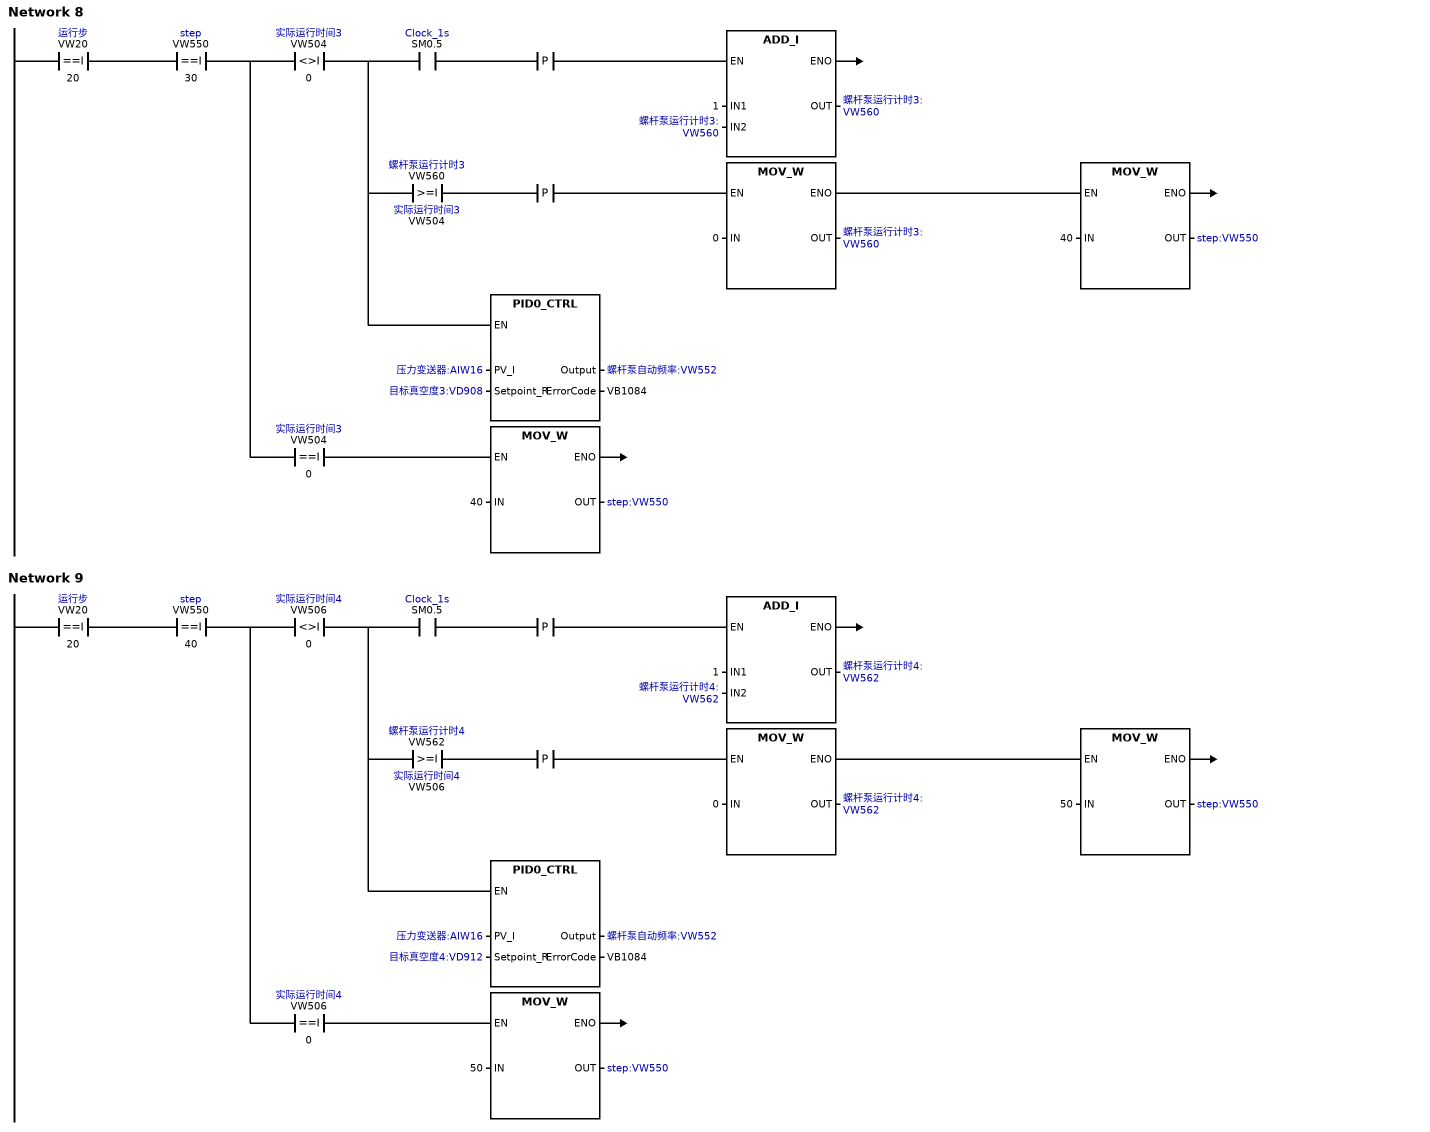
Network 8
LDW=   运行步:VW20, 20
AW=    step:VW550, 30
LPS
AW<>   实际运行时间3:VW504, 0
LPS
A      Clock_1s:SM0.5
EU
+I     1, 螺杆泵运行计时3:VW560
LRD
AW>=   螺杆泵运行计时3:VW560, 实际运行时间3:VW504
EU
MOVW   0, 螺杆泵运行计时3:VW560
AENO
MOVW   40, step:VW550
LPP
CALL   PID0_CTRL:SBR10, 压力变送器:AIW16, 目标真空度3:VD908, 螺杆泵自动频率:VW552, VB1084
LPP
AW=    实际运行时间3:VW504, 0
MOVW   40, step:VW550
Network 9
LDW=   运行步:VW20, 20
AW=    step:VW550, 40
LPS
AW<>   实际运行时间4:VW506, 0
LPS
A      Clock_1s:SM0.5
EU
+I     1, 螺杆泵运行计时4:VW562
LRD
AW>=   螺杆泵运行计时4:VW562, 实际运行时间4:VW506
EU
MOVW   0, 螺杆泵运行计时4:VW562
AENO
MOVW   50, step:VW550
LPP
CALL   PID0_CTRL:SBR10, 压力变送器:AIW16, 目标真空度4:VD912, 螺杆泵自动频率:VW552, VB1084
LPP
AW=    实际运行时间4:VW506, 0
MOVW   50, step:VW550
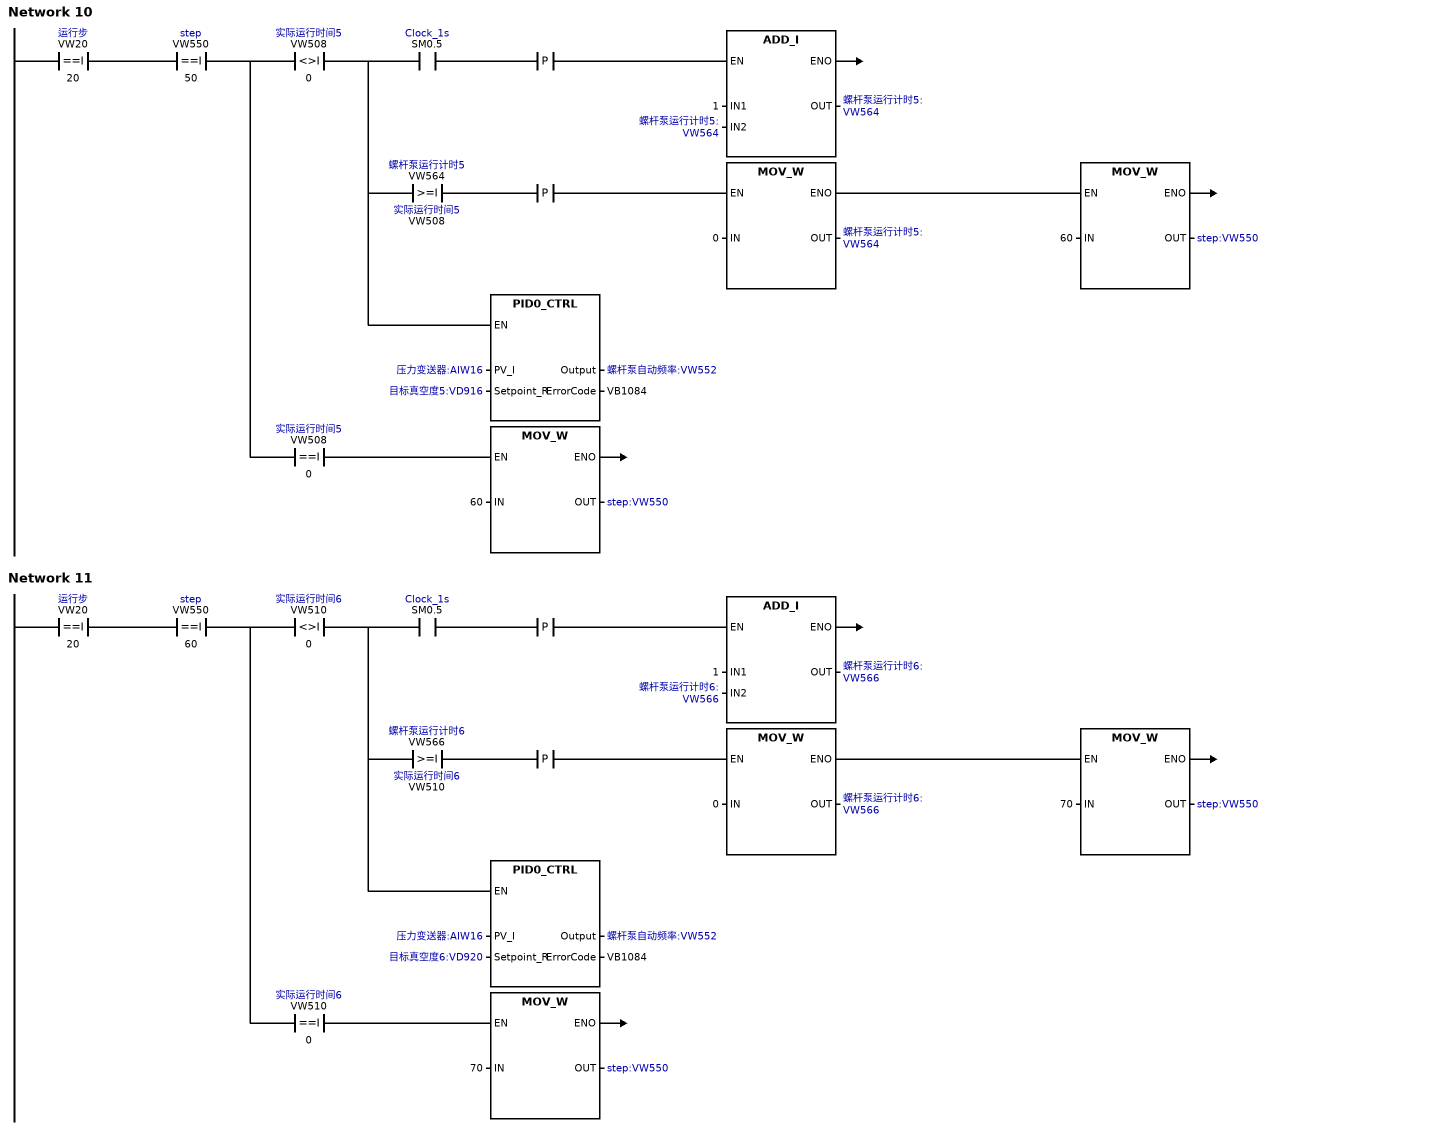
Network 10
LDW=   运行步:VW20, 20
AW=    step:VW550, 50
LPS
AW<>   实际运行时间5:VW508, 0
LPS
A      Clock_1s:SM0.5
EU
+I     1, 螺杆泵运行计时5:VW564
LRD
AW>=   螺杆泵运行计时5:VW564, 实际运行时间5:VW508
EU
MOVW   0, 螺杆泵运行计时5:VW564
AENO
MOVW   60, step:VW550
LPP
CALL   PID0_CTRL:SBR10, 压力变送器:AIW16, 目标真空度5:VD916, 螺杆泵自动频率:VW552, VB1084
LPP
AW=    实际运行时间5:VW508, 0
MOVW   60, step:VW550
Network 11
LDW=   运行步:VW20, 20
AW=    step:VW550, 60
LPS
AW<>   实际运行时间6:VW510, 0
LPS
A      Clock_1s:SM0.5
EU
+I     1, 螺杆泵运行计时6:VW566
LRD
AW>=   螺杆泵运行计时6:VW566, 实际运行时间6:VW510
EU
MOVW   0, 螺杆泵运行计时6:VW566
AENO
MOVW   70, step:VW550
LPP
CALL   PID0_CTRL:SBR10, 压力变送器:AIW16, 目标真空度6:VD920, 螺杆泵自动频率:VW552, VB1084
LPP
AW=    实际运行时间6:VW510, 0
MOVW   70, step:VW550
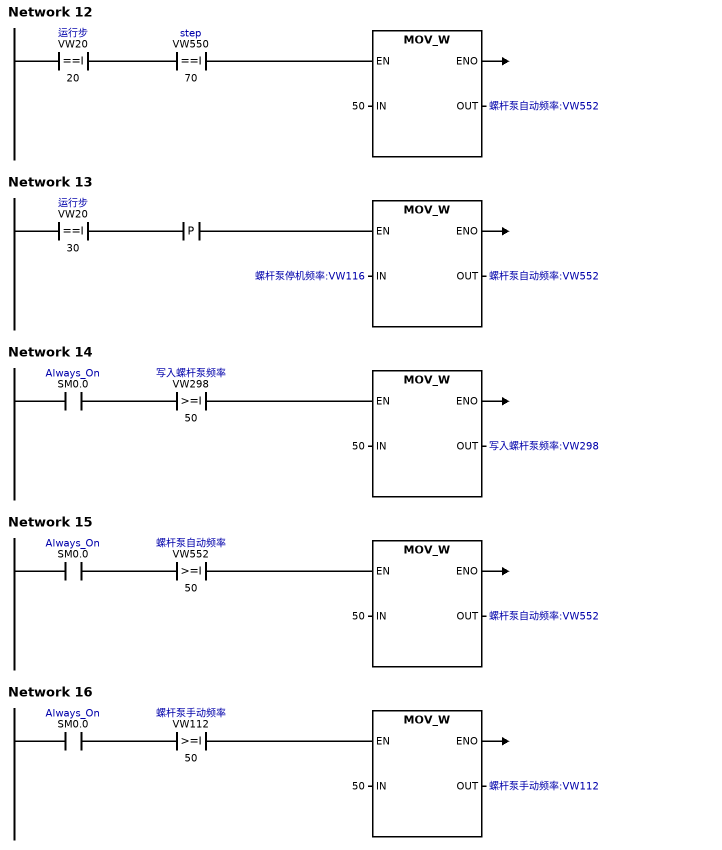
Network 12
LDW=   运行步:VW20, 20
AW=    step:VW550, 70
MOVW   50, 螺杆泵自动频率:VW552
Network 13
LDW=   运行步:VW20, 30
EU
MOVW   螺杆泵停机频率:VW116, 螺杆泵自动频率:VW552
Network 14
LD     Always_On:SM0.0
AW>=   写入螺杆泵频率:VW298, 50
MOVW   50, 写入螺杆泵频率:VW298
Network 15
LD     Always_On:SM0.0
AW>=   螺杆泵自动频率:VW552, 50
MOVW   50, 螺杆泵自动频率:VW552
Network 16
LD     Always_On:SM0.0
AW>=   螺杆泵手动频率:VW112, 50
MOVW   50, 螺杆泵手动频率:VW112
END_SUBROUTINE_BLOCK

// SBR16: protected block, not included

// SBR17: protected block, not included

DATA_BLOCK_TAB 页面_1
BEGIN
//数据页注释
//按 F1 获取帮助和示例数据页
         冷却水温度报警值, 45.0
         冷却水温度停机值, 55.0
         预设清洗时间, 300
         预设吹扫时间, 300
         罗茨泵运行真空度1, 10.0
         罗茨泵运行真空度2, 6.0
         罗茨泵停止真空度1, 12.0
         罗茨泵停止真空度2, 9.0
         螺杆泵手动频率, 50
         罗茨泵手动频率, 50
         罗茨泵手动频率2, 50
         螺杆泵停机频率, 30
         预设冷却水关闭时间, 600
         排液间隔时间, 20
END_DATA_BLOCK_TAB
